// TIA Portal V17 export
// export: Created 2025-03-12T15:35:17.3302605Z, ExportSetting WithDefaults, DisplayName Totally Integrated Automation Portal, DisplayVersion V17 Update 8, DisplayName TIA Portal Openness, DisplayVersion V17 Update 8, DisplayName TIA Portal Version Control Interface, DisplayVersion V17, DisplayName SINAMICS Startdrive Advanced, DisplayVersion V17 SP2, DisplayName SINAMICS Startdrive G110M, G120, G120C, G120D, G120P, G115D, DisplayVersion V17 SP2, DisplayName SINAMICS Startdrive G130, G150, S120, S150, SINAMICS MV, S210, DisplayVersion V17 SP2, DisplayName STEP 7 Professional, DisplayVersion V17 Update 8, DisplayName SINUMERIK ONE STEP 7 Toolbox, DisplayVersion V17 Update 12, DisplayName SINUMERIK 840D sl STEP 7 Toolbox, DisplayVersion V17 Update 12, DisplayName STEP 7 Safety, DisplayVersion V17 Update 6, DisplayName WinCC Advanced, DisplayVersion V17 Update 8
DATA_BLOCK "DB138_CLADDING_AXIS_X13"   // DB138
{ DB_Accessible_From_OPC_UA := 'FALSE' }
AUTHOR : ETXETAR
VERSION : 1.0
// stored: AutoNumber false, DBAccessibleFromOPCUA false, DBAccessibleFromWebserver true, InstanceOfName FB32_AXIS, InstanceOfType FB
"FB32_AXIS"
   // VAR_INPUT
   //    OPTIONS_0 : Byte := 16#00;
   //    OPTIONS_1 : Byte := 16#00;
   //    SAFETY_BYPASS : Bool := FALSE;
   //    OPTIMIZATION_BYPASS : Bool := FALSE;
   //    AX_ENABLE : Bool := TRUE;
   //    TEST_STOP_BRAKE_TEST_AX_NUM : Bool := FALSE;
   //    PARAMETER_SET_0 : Bool := TRUE;
   //    PARAMETER_SET_1 : Bool := FALSE;
   //    PARAMETER_SET_2 : Bool := FALSE;
   //    PARAMETER_SET_3 : Bool := FALSE;
   //    MOVE_AXIS : Bool := FALSE;
   //    SAFE_ENABLED : Bool := TRUE;
   //    FEED_HOLD_COND : Bool := FALSE;
   //    AX_TORQUE_ENABLE : Bool := FALSE;
   //    MPP_AXIS_SELECTED : Bool := FALSE;
   //    HMI_AXIS_SELECTED : Bool := FALSE;
   //    HMI_REQ_LINE : Bool := FALSE;
   //    JOG_MINUS_REQ_NOT_FC18 : Bool := FALSE;
   //    JOG_PLUS_REQ_NOT_FC18 : Bool := FALSE;
   //    JOG_MINUS_REQ_FC18 : Bool := FALSE;
   //    JOG_PLUS_REQ_FC18 : Bool := FALSE;
   //    FC18_EXTERNAL_POS : Real := 0.0;
   //    AUTO_RETURN_COMMAND : Bool := FALSE;
   //    AUTO_ADVANCE_COMMAND : Bool := FALSE;
   //    DELETE_DISTANCE_TO_GO : Bool := FALSE;
   //    FEED_OVERRIDE : Byte := 16#01;
   //    FEED_OVER_ACTIVE : Bool := TRUE;
   //    READ_POS : DWord := 16#C391_0000;
   //    UNIT_ALARM : UInt := 1;
   //    STATION_ALARM : UInt := 0;
   // END_VAR
   // VAR_OUTPUT
   //    MOTOR_ACTIVE : Bool := TRUE;
   //    MOVE_AX : Bool := TRUE;
   //    FEED_HOLD_CONDITIONS : Bool := FALSE;
   //    ACTIVE_PARAMETER_SET : Byte := 16#01;
   //    AX_NOT_REFERENCE_ALM : Bool := FALSE;
   //    AX_B_NOT_IN_PST_180_90_ALM : Bool := FALSE;
   //    MAST_SLAVE_MODE_NOT_ACTIV_ALM : Bool := FALSE;
   //    AX_TORQUE_EXCEEDED_ALM : Bool := FALSE;
   //    AXIS_POS : Real := -290.0;
   //    HMI_MOTION_EXECUTABILITY_LEFT : Bool := FALSE;
   //    HMI_MOTION_EXECUTABILITY_RIGHT : Bool := FALSE;
   //    HMI_MOTION_END_POS_LEFT : Bool := FALSE;
   //    HMI_MOTION_END_POS_RIGHT : Bool := FALSE;
   //    HMI_MOTION_ACTIVE_LEFT : Bool := FALSE;
   //    HMI_MOTION_ACTIVE_RIGHT : Bool := FALSE;
   // END_VAR
   // VAR_IN_OUT
   //    AxisDB : "LBP_typeAxisX";
   // END_VAR
   // VAR RETAIN
   //    AXIS { S7_SetPoint := 'True'} : "AXIS";
   //    TIMER_PULSES_ENABLE { S7_SetPoint := 'True'} : TOF_TIME;
   //    SAFETY_POSITIONS { S7_SetPoint := 'True'} : "FB33_SAFETY_POSITIONS";
   // END_VAR
BEGIN
   AXIS.ENABLED := TRUE;
   AXIS.SELECTED := FALSE;
   AXIS.HMI_JOG_MINUS_RQ := FALSE;
   AXIS.HMI_JOG_PLUS_RQ := FALSE;
   AXIS.HMI_JOG_MINUS_CMM := FALSE;
   AXIS.HMI_JOG_PLUS_CMM := FALSE;
   AXIS.AUTO_RETURN_CMM := FALSE;
   AXIS.AUTO_ADVANCE_CMM := FALSE;
   AXIS.JOG_HELP := FALSE;
   AXIS.MINUS_BUTTON_HELP := FALSE;
   AXIS.PLUS_BUTTON_HELP := FALSE;
   AXIS.OPERATOR_HELP := FALSE;
   AXIS.P1_TRIGGER := FALSE;
   AXIS.P2_TRIGGER := FALSE;
   AXIS.N1_TRIGGER := FALSE;
   AXIS.N2_TRIGGER := FALSE;
   AXIS.POS_TO_GO_FC18 := 0.0;
   AXIS.FC18_AXIS_IN_POS := FALSE;
   AXIS.FC18_FAULT := FALSE;
   AXIS.E_GANT_GROUP_SYN := FALSE;
   TIMER_PULSES_ENABLE.PT := T#1S;
   TIMER_PULSES_ENABLE.IN := TRUE;
   SAFETY_POSITIONS.MEAS_SYS_1_ACTIVE_REFERENCED := TRUE;
   SAFETY_POSITIONS.MEAS_SYS_2_ACTIVE_REFERENCED := FALSE;
   SAFETY_POSITIONS.AXIS_POS := -290.0;
   SAFETY_POSITIONS.AX_POS_0_DEGREES.TOLERANCE := 0.005;
   SAFETY_POSITIONS.AX_POS_0_DEGREES.POSITION_0_TOLERANCE_PLUS := 0.005;
   SAFETY_POSITIONS.AX_POS_0_DEGREES.POSITION_0_TOLERANCE_MINUS := -0.005;
   SAFETY_POSITIONS.AX_POS_0_DEGREES.POSITION_360_TOLERANCE_PLUS := 360.005;
   SAFETY_POSITIONS.AX_POS_0_DEGREES.POSITION_360_TOLERANCE_MINUS := 359.995;
   SAFETY_POSITIONS.AX_POS_0_DEGREES.IN_POSITION := FALSE;
   SAFETY_POSITIONS.AX_POS_90_DEGREES.TOLERANCE := 0.005;
   SAFETY_POSITIONS.AX_POS_90_DEGREES.POSITION_TOLERANCE_PLUS := 90.005;
   SAFETY_POSITIONS.AX_POS_90_DEGREES.POSITION_TOLERANCE_MINUS := 89.995;
   SAFETY_POSITIONS.AX_POS_90_DEGREES.IN_POSITION := FALSE;
   SAFETY_POSITIONS.AX_POS_180_DEGREES.TOLERANCE := 0.005;
   SAFETY_POSITIONS.AX_POS_180_DEGREES.POSITION_TOLERANCE_PLUS := 180.005;
   SAFETY_POSITIONS.AX_POS_180_DEGREES.POSITION_TOLERANCE_MINUS := 179.995;
   SAFETY_POSITIONS.AX_POS_180_DEGREES.IN_POSITION := FALSE;
   SAFETY_POSITIONS.AX_POS_270_DEGREES.TOLERANCE := 0.005;
   SAFETY_POSITIONS.AX_POS_270_DEGREES.POSITION_TOLERANCE_PLUS := 270.005;
   SAFETY_POSITIONS.AX_POS_270_DEGREES.POSITION_TOLERANCE_MINUS := 269.995;
   SAFETY_POSITIONS.AX_POS_270_DEGREES.IN_POSITION := FALSE;
   SAFETY_POSITIONS.AX_POS_MINUS_90_DEGREES := FALSE;
   SAFETY_POSITIONS.AX_POS_MINUS_180_DEGREES := FALSE;
   SAFETY_POSITIONS.AX_POS_MINUS_270_DEGREES := FALSE;
   SAFETY_POSITIONS.SAFETY_POSITION_1.HMI_POSITION := -290.0;
   SAFETY_POSITIONS.SAFETY_POSITION_1.TOLERANCE_PLUS := 0.01;
   SAFETY_POSITIONS.SAFETY_POSITION_1.TOLERANCE_MINUS := 0.01;
   SAFETY_POSITIONS.SAFETY_POSITION_1.POSITION_TOLERANCE_PLUS := -289.99;
   SAFETY_POSITIONS.SAFETY_POSITION_1.POSITION_TOLERANCE_MINUS := -290.01;
   SAFETY_POSITIONS.SAFETY_POSITION_1.IN_POSITION := TRUE;
   SAFETY_POSITIONS.SAFETY_POSITION_1.GREATER_TOLERANCE_PLUS := FALSE;
   SAFETY_POSITIONS.SAFETY_POSITION_1.GREATER_TOLERANCE_MINUS := TRUE;
   SAFETY_POSITIONS.SAFETY_POSITION_1.LOWER_TOLERANCE_PLUS := TRUE;
   SAFETY_POSITIONS.SAFETY_POSITION_1.LOWER_TOLERANCE_MINUS := FALSE;
   SAFETY_POSITIONS.SAFETY_POSITION_2.HMI_POSITION := 1.1;
   SAFETY_POSITIONS.SAFETY_POSITION_2.TOLERANCE_PLUS := 0.01;
   SAFETY_POSITIONS.SAFETY_POSITION_2.TOLERANCE_MINUS := 0.01;
   SAFETY_POSITIONS.SAFETY_POSITION_2.POSITION_TOLERANCE_PLUS := 1.11;
   SAFETY_POSITIONS.SAFETY_POSITION_2.POSITION_TOLERANCE_MINUS := 1.09;
   SAFETY_POSITIONS.SAFETY_POSITION_2.IN_POSITION := FALSE;
   SAFETY_POSITIONS.SAFETY_POSITION_2.GREATER_TOLERANCE_PLUS := FALSE;
   SAFETY_POSITIONS.SAFETY_POSITION_2.GREATER_TOLERANCE_MINUS := FALSE;
   SAFETY_POSITIONS.SAFETY_POSITION_2.LOWER_TOLERANCE_PLUS := FALSE;
   SAFETY_POSITIONS.SAFETY_POSITION_2.LOWER_TOLERANCE_MINUS := FALSE;
   SAFETY_POSITIONS.SAFETY_POSITION_3.HMI_POSITION := 1.1;
   SAFETY_POSITIONS.SAFETY_POSITION_3.TOLERANCE_PLUS := 0.01;
   SAFETY_POSITIONS.SAFETY_POSITION_3.TOLERANCE_MINUS := 0.01;
   SAFETY_POSITIONS.SAFETY_POSITION_3.POSITION_TOLERANCE_PLUS := 1.11;
   SAFETY_POSITIONS.SAFETY_POSITION_3.POSITION_TOLERANCE_MINUS := 1.09;
   SAFETY_POSITIONS.SAFETY_POSITION_3.IN_POSITION := FALSE;
   SAFETY_POSITIONS.SAFETY_POSITION_3.GREATER_TOLERANCE_PLUS := FALSE;
   SAFETY_POSITIONS.SAFETY_POSITION_3.GREATER_TOLERANCE_MINUS := FALSE;
   SAFETY_POSITIONS.SAFETY_POSITION_3.LOWER_TOLERANCE_PLUS := FALSE;
   SAFETY_POSITIONS.SAFETY_POSITION_3.LOWER_TOLERANCE_MINUS := FALSE;
   SAFETY_POSITIONS.SAFETY_POSITION_4.HMI_POSITION := 1.1;
   SAFETY_POSITIONS.SAFETY_POSITION_4.TOLERANCE_PLUS := 0.01;
   SAFETY_POSITIONS.SAFETY_POSITION_4.TOLERANCE_MINUS := 0.01;
   SAFETY_POSITIONS.SAFETY_POSITION_4.POSITION_TOLERANCE_PLUS := 1.11;
   SAFETY_POSITIONS.SAFETY_POSITION_4.POSITION_TOLERANCE_MINUS := 1.09;
   SAFETY_POSITIONS.SAFETY_POSITION_4.IN_POSITION := FALSE;
   SAFETY_POSITIONS.SAFETY_POSITION_4.GREATER_TOLERANCE_PLUS := FALSE;
   SAFETY_POSITIONS.SAFETY_POSITION_4.GREATER_TOLERANCE_MINUS := FALSE;
   SAFETY_POSITIONS.SAFETY_POSITION_4.LOWER_TOLERANCE_PLUS := FALSE;
   SAFETY_POSITIONS.SAFETY_POSITION_4.LOWER_TOLERANCE_MINUS := FALSE;
   SAFETY_POSITIONS.SAFETY_POSITION_5.HMI_POSITION := 1.1;
   SAFETY_POSITIONS.SAFETY_POSITION_5.TOLERANCE_PLUS := 0.01;
   SAFETY_POSITIONS.SAFETY_POSITION_5.TOLERANCE_MINUS := 0.01;
   SAFETY_POSITIONS.SAFETY_POSITION_5.POSITION_TOLERANCE_PLUS := 1.11;
   SAFETY_POSITIONS.SAFETY_POSITION_5.POSITION_TOLERANCE_MINUS := 1.09;
   SAFETY_POSITIONS.SAFETY_POSITION_5.IN_POSITION := FALSE;
   SAFETY_POSITIONS.SAFETY_POSITION_5.GREATER_TOLERANCE_PLUS := FALSE;
   SAFETY_POSITIONS.SAFETY_POSITION_5.GREATER_TOLERANCE_MINUS := FALSE;
   SAFETY_POSITIONS.SAFETY_POSITION_5.LOWER_TOLERANCE_PLUS := FALSE;
   SAFETY_POSITIONS.SAFETY_POSITION_5.LOWER_TOLERANCE_MINUS := FALSE;
   SAFETY_POSITIONS.SAFETY_POSITION_6.HMI_POSITION := 1.1;
   SAFETY_POSITIONS.SAFETY_POSITION_6.TOLERANCE_PLUS := 0.01;
   SAFETY_POSITIONS.SAFETY_POSITION_6.TOLERANCE_MINUS := 0.01;
   SAFETY_POSITIONS.SAFETY_POSITION_6.POSITION_TOLERANCE_PLUS := 1.11;
   SAFETY_POSITIONS.SAFETY_POSITION_6.POSITION_TOLERANCE_MINUS := 1.09;
   SAFETY_POSITIONS.SAFETY_POSITION_6.IN_POSITION := FALSE;
   SAFETY_POSITIONS.SAFETY_POSITION_6.GREATER_TOLERANCE_PLUS := FALSE;
   SAFETY_POSITIONS.SAFETY_POSITION_6.GREATER_TOLERANCE_MINUS := FALSE;
   SAFETY_POSITIONS.SAFETY_POSITION_6.LOWER_TOLERANCE_PLUS := FALSE;
   SAFETY_POSITIONS.SAFETY_POSITION_6.LOWER_TOLERANCE_MINUS := FALSE;
   SAFETY_POSITIONS.SAFETY_POSITION_7.HMI_POSITION := 1.1;
   SAFETY_POSITIONS.SAFETY_POSITION_7.TOLERANCE_PLUS := 0.01;
   SAFETY_POSITIONS.SAFETY_POSITION_7.TOLERANCE_MINUS := 0.01;
   SAFETY_POSITIONS.SAFETY_POSITION_7.POSITION_TOLERANCE_PLUS := 1.11;
   SAFETY_POSITIONS.SAFETY_POSITION_7.POSITION_TOLERANCE_MINUS := 1.09;
   SAFETY_POSITIONS.SAFETY_POSITION_7.IN_POSITION := FALSE;
   SAFETY_POSITIONS.SAFETY_POSITION_7.GREATER_TOLERANCE_PLUS := FALSE;
   SAFETY_POSITIONS.SAFETY_POSITION_7.GREATER_TOLERANCE_MINUS := FALSE;
   SAFETY_POSITIONS.SAFETY_POSITION_7.LOWER_TOLERANCE_PLUS := FALSE;
   SAFETY_POSITIONS.SAFETY_POSITION_7.LOWER_TOLERANCE_MINUS := FALSE;
   SAFETY_POSITIONS.SAFETY_POSITION_8.HMI_POSITION := 1.1;
   SAFETY_POSITIONS.SAFETY_POSITION_8.TOLERANCE_PLUS := 0.01;
   SAFETY_POSITIONS.SAFETY_POSITION_8.TOLERANCE_MINUS := 0.01;
   SAFETY_POSITIONS.SAFETY_POSITION_8.POSITION_TOLERANCE_PLUS := 1.11;
   SAFETY_POSITIONS.SAFETY_POSITION_8.POSITION_TOLERANCE_MINUS := 1.09;
   SAFETY_POSITIONS.SAFETY_POSITION_8.IN_POSITION := FALSE;
   SAFETY_POSITIONS.SAFETY_POSITION_8.GREATER_TOLERANCE_PLUS := FALSE;
   SAFETY_POSITIONS.SAFETY_POSITION_8.GREATER_TOLERANCE_MINUS := FALSE;
   SAFETY_POSITIONS.SAFETY_POSITION_8.LOWER_TOLERANCE_PLUS := FALSE;
   SAFETY_POSITIONS.SAFETY_POSITION_8.LOWER_TOLERANCE_MINUS := FALSE;
   SAFETY_POSITIONS.SAFETY_POSITION_9.HMI_POSITION := 1.1;
   SAFETY_POSITIONS.SAFETY_POSITION_9.TOLERANCE_PLUS := 0.01;
   SAFETY_POSITIONS.SAFETY_POSITION_9.TOLERANCE_MINUS := 0.01;
   SAFETY_POSITIONS.SAFETY_POSITION_9.POSITION_TOLERANCE_PLUS := 1.11;
   SAFETY_POSITIONS.SAFETY_POSITION_9.POSITION_TOLERANCE_MINUS := 1.09;
   SAFETY_POSITIONS.SAFETY_POSITION_9.IN_POSITION := FALSE;
   SAFETY_POSITIONS.SAFETY_POSITION_9.GREATER_TOLERANCE_PLUS := FALSE;
   SAFETY_POSITIONS.SAFETY_POSITION_9.GREATER_TOLERANCE_MINUS := FALSE;
   SAFETY_POSITIONS.SAFETY_POSITION_9.LOWER_TOLERANCE_PLUS := FALSE;
   SAFETY_POSITIONS.SAFETY_POSITION_9.LOWER_TOLERANCE_MINUS := FALSE;
   SAFETY_POSITIONS.SAFETY_POSITION_10.HMI_POSITION := 1.1;
   SAFETY_POSITIONS.SAFETY_POSITION_10.TOLERANCE_PLUS := 0.01;
   SAFETY_POSITIONS.SAFETY_POSITION_10.TOLERANCE_MINUS := 0.01;
   SAFETY_POSITIONS.SAFETY_POSITION_10.POSITION_TOLERANCE_PLUS := 1.11;
   SAFETY_POSITIONS.SAFETY_POSITION_10.POSITION_TOLERANCE_MINUS := 1.09;
   SAFETY_POSITIONS.SAFETY_POSITION_10.IN_POSITION := FALSE;
   SAFETY_POSITIONS.SAFETY_POSITION_10.GREATER_TOLERANCE_PLUS := FALSE;
   SAFETY_POSITIONS.SAFETY_POSITION_10.GREATER_TOLERANCE_MINUS := FALSE;
   SAFETY_POSITIONS.SAFETY_POSITION_10.LOWER_TOLERANCE_PLUS := FALSE;
   SAFETY_POSITIONS.SAFETY_POSITION_10.LOWER_TOLERANCE_MINUS := FALSE;
END_DATA_BLOCK
